{attribute 'qualified_only'}
{attribute 'strict'}
TYPE DUT :
(
	enum_member := 0
);
END_TYPE

(* stored: Version 1.1.0.1, ProductVersion 3.1.4024.15
   DUT DUT: Id {db029942-4cc1-4176-b7f1-3b5be71beb89} *)
